(*======================================================================================================================================*)
(*fb_StringConvRB16F:	Zusammensetzen des Strings für 16Fach Bus Relaismodul		*)
(*
Date          	| Version    	| created under        	| Author          	| Remark *)
(*====================================================================================================================================================*)
(*08/05/2025   	| 1.00      		| TC3		  		| N.Kersting       | first release *)
(*====================================================================================================================================================*)
FUNCTION_BLOCK fb_StringConvRB16F
VAR_INPUT
	I_bReset			:BOOL;							(* Reset Befehl auslösen *)
	I_bRedLEDOn			:BOOL;							(* Schaltet nur die Rote Modul LED ein*)
	I_bRedLEDOff		:BOOL;							(* Schaltet nur die Rote Modul LED aus*)
	I_diID				:DINT;							(* Device ID *)
	I_bOut    	 		:ARRAY[1..16] OF BOOL;     	  	(* gewünschter Relais zustand (TRUE = An %)*)
	
	I_iSection			:INT :=1;							(* Paarweise Schalten 1= 1&2 2= 3&4 usw. *)
	
	I_sStartZeichen		:BYTE := 16#FD;					(* Startzeichen Präfix *)
	I_sEndZeichen		:BYTE := 16#FE;					(* Endzeichen Suffix *)
END_VAR
VAR_OUTPUT
	Q_sConvString		:STRING(255);
END_VAR
VAR
	iStartOut			:INT := 1;
	iStartInstIDExt		:INT :=65;
	
END_VAR

IF NOT I_bReset
THEN
	IF I_bRedLEDOn
	THEN
		(* Rote Modul LED Ein*)
		iStartInstIDExt := 210;
		
		Q_sConvString:=	CONCAT(F_ToCHR(I_sStartZeichen),DINT_TO_STRING(I_diID));
		Q_sConvString:=	CONCAT(Q_sConvString,'.OUT.');
		Q_sConvString:=	CONCAT(Q_sConvString,INT_TO_STRING(iStartInstIDExt));
		Q_sConvString:=	CONCAT(Q_sConvString,'.ON');
		Q_sConvString:=	CONCAT(Q_sConvString,F_ToCHR(I_sEndZeichen));
	ELSIF
		I_bRedLEDOff
	THEN
		(* Rote Modul LED Aus*)
		iStartInstIDExt := 210;
		
		Q_sConvString:=	CONCAT(F_ToCHR(I_sStartZeichen),DINT_TO_STRING(I_diID));
		Q_sConvString:=	CONCAT(Q_sConvString,'.OUT.');
		Q_sConvString:=	CONCAT(Q_sConvString,INT_TO_STRING(iStartInstIDExt));
		Q_sConvString:=	CONCAT(Q_sConvString,'.OFF');
		Q_sConvString:=	CONCAT(Q_sConvString,F_ToCHR(I_sEndZeichen));
	ELSE
		CASE I_iSection OF
			
		0:	Q_sConvString:='';
		
		1:	(* 1 & 2 Schalten *)
			iStartInstIDExt := 17;
			iStartOut :=	1;
			
			Q_sConvString:=	CONCAT(F_ToCHR(I_sStartZeichen),DINT_TO_STRING(I_diID));
			Q_sConvString:=	CONCAT(Q_sConvString,'.OUT.');
			Q_sConvString:=	CONCAT(Q_sConvString,INT_TO_STRING(iStartInstIDExt));
			IF I_bOut[iStartOut]
			THEN
				Q_sConvString:=	CONCAT(Q_sConvString,'.ON');
			ELSE
				Q_sConvString:=	CONCAT(Q_sConvString,'.OFF');
			END_IF
			Q_sConvString:=	CONCAT(Q_sConvString,F_ToCHR(I_sEndZeichen));
			
			(* ##2 ##*)
			iStartInstIDExt := iStartInstIDExt +1;
			iStartOut:= iStartOut+1;
			
			Q_sConvString:=	CONCAT(Q_sConvString,F_ToCHR(I_sStartZeichen));
			Q_sConvString:=	CONCAT(Q_sConvString,DINT_TO_STRING(I_diID));
			Q_sConvString:=	CONCAT(Q_sConvString,'.OUT.');
			Q_sConvString:=	CONCAT(Q_sConvString,INT_TO_STRING(iStartInstIDExt));
			IF I_bOut[iStartOut]
			THEN
				Q_sConvString:=	CONCAT(Q_sConvString,'.ON');
			ELSE
				Q_sConvString:=	CONCAT(Q_sConvString,'.OFF');
			END_IF
			Q_sConvString:=	CONCAT(Q_sConvString,F_ToCHR(I_sEndZeichen));
		
			(* ##3 ##*)
			iStartInstIDExt := iStartInstIDExt +1;
			iStartOut:= iStartOut+1;
			
			Q_sConvString:=	CONCAT(Q_sConvString,F_ToCHR(I_sStartZeichen));
			Q_sConvString:=	CONCAT(Q_sConvString,DINT_TO_STRING(I_diID));
			Q_sConvString:=	CONCAT(Q_sConvString,'.OUT.');
			Q_sConvString:=	CONCAT(Q_sConvString,INT_TO_STRING(iStartInstIDExt));
			IF I_bOut[iStartOut]
			THEN
				Q_sConvString:=	CONCAT(Q_sConvString,'.ON');
			ELSE
				Q_sConvString:=	CONCAT(Q_sConvString,'.OFF');
			END_IF
			Q_sConvString:=	CONCAT(Q_sConvString,F_ToCHR(I_sEndZeichen));
			
			(* ##4 ##*)
			iStartInstIDExt := iStartInstIDExt +1;
			iStartOut:= iStartOut+1;
			
			Q_sConvString:=	CONCAT(Q_sConvString,F_ToCHR(I_sStartZeichen));
			Q_sConvString:=	CONCAT(Q_sConvString,DINT_TO_STRING(I_diID));
			Q_sConvString:=	CONCAT(Q_sConvString,'.OUT.');
			Q_sConvString:=	CONCAT(Q_sConvString,INT_TO_STRING(iStartInstIDExt));
			IF I_bOut[iStartOut]
			THEN
				Q_sConvString:=	CONCAT(Q_sConvString,'.ON');
			ELSE
				Q_sConvString:=	CONCAT(Q_sConvString,'.OFF');
			END_IF
			Q_sConvString:=	CONCAT(Q_sConvString,F_ToCHR(I_sEndZeichen));
		
			(* ##5 ##*)
			iStartInstIDExt := iStartInstIDExt +1;
			iStartOut:= iStartOut+1;
			
			Q_sConvString:=	CONCAT(Q_sConvString,F_ToCHR(I_sStartZeichen));
			Q_sConvString:=	CONCAT(Q_sConvString,DINT_TO_STRING(I_diID));
			Q_sConvString:=	CONCAT(Q_sConvString,'.OUT.');
			Q_sConvString:=	CONCAT(Q_sConvString,INT_TO_STRING(iStartInstIDExt));
			IF I_bOut[iStartOut]
			THEN
				Q_sConvString:=	CONCAT(Q_sConvString,'.ON');
			ELSE
				Q_sConvString:=	CONCAT(Q_sConvString,'.OFF');
			END_IF
			Q_sConvString:=	CONCAT(Q_sConvString,F_ToCHR(I_sEndZeichen));
			
			(* ##6 ##*)
			iStartInstIDExt := iStartInstIDExt +1;
			iStartOut:= iStartOut+1;
			
			Q_sConvString:=	CONCAT(Q_sConvString,F_ToCHR(I_sStartZeichen));
			Q_sConvString:=	CONCAT(Q_sConvString,DINT_TO_STRING(I_diID));
			Q_sConvString:=	CONCAT(Q_sConvString,'.OUT.');
			Q_sConvString:=	CONCAT(Q_sConvString,INT_TO_STRING(iStartInstIDExt));
			IF I_bOut[iStartOut]
			THEN
				Q_sConvString:=	CONCAT(Q_sConvString,'.ON');
			ELSE
				Q_sConvString:=	CONCAT(Q_sConvString,'.OFF');
			END_IF
			Q_sConvString:=	CONCAT(Q_sConvString,F_ToCHR(I_sEndZeichen));
		
			(* ##7 ##*)
			iStartInstIDExt := iStartInstIDExt +1;
			iStartOut:= iStartOut+1;
			
			Q_sConvString:=	CONCAT(Q_sConvString,F_ToCHR(I_sStartZeichen));
			Q_sConvString:=	CONCAT(Q_sConvString,DINT_TO_STRING(I_diID));
			Q_sConvString:=	CONCAT(Q_sConvString,'.OUT.');
			Q_sConvString:=	CONCAT(Q_sConvString,INT_TO_STRING(iStartInstIDExt));
			IF I_bOut[iStartOut]
			THEN
				Q_sConvString:=	CONCAT(Q_sConvString,'.ON');
			ELSE
				Q_sConvString:=	CONCAT(Q_sConvString,'.OFF');
			END_IF
			Q_sConvString:=	CONCAT(Q_sConvString,F_ToCHR(I_sEndZeichen));
			
			(* ##8 ##*)
			iStartInstIDExt := iStartInstIDExt +1;
			iStartOut:= iStartOut+1;
			
			Q_sConvString:=	CONCAT(Q_sConvString,F_ToCHR(I_sStartZeichen));
			Q_sConvString:=	CONCAT(Q_sConvString,DINT_TO_STRING(I_diID));
			Q_sConvString:=	CONCAT(Q_sConvString,'.OUT.');
			Q_sConvString:=	CONCAT(Q_sConvString,INT_TO_STRING(iStartInstIDExt));
			IF I_bOut[iStartOut]
			THEN
				Q_sConvString:=	CONCAT(Q_sConvString,'.ON');
			ELSE
				Q_sConvString:=	CONCAT(Q_sConvString,'.OFF');
			END_IF
			Q_sConvString:=	CONCAT(Q_sConvString,F_ToCHR(I_sEndZeichen));
		
		2:	(* 9 & 10 Schalten *)
			iStartInstIDExt := 33;
			iStartOut :=	9;
			
			Q_sConvString:=	CONCAT(F_ToCHR(I_sStartZeichen),DINT_TO_STRING(I_diID));
			Q_sConvString:=	CONCAT(Q_sConvString,'.OUT.');
			Q_sConvString:=	CONCAT(Q_sConvString,INT_TO_STRING(iStartInstIDExt));
			IF I_bOut[iStartOut]
			THEN
				Q_sConvString:=	CONCAT(Q_sConvString,'.ON');
			ELSE
				Q_sConvString:=	CONCAT(Q_sConvString,'.OFF');
			END_IF
			Q_sConvString:=	CONCAT(Q_sConvString,F_ToCHR(I_sEndZeichen));
			
			(* ##10 ##*)
			iStartInstIDExt := iStartInstIDExt +1;
			iStartOut:= iStartOut+1;
			
			Q_sConvString:=	CONCAT(Q_sConvString,F_ToCHR(I_sStartZeichen));
			Q_sConvString:=	CONCAT(Q_sConvString,DINT_TO_STRING(I_diID));
			Q_sConvString:=	CONCAT(Q_sConvString,'.OUT.');
			Q_sConvString:=	CONCAT(Q_sConvString,INT_TO_STRING(iStartInstIDExt));
			IF I_bOut[iStartOut]
			THEN
				Q_sConvString:=	CONCAT(Q_sConvString,'.ON');
			ELSE
				Q_sConvString:=	CONCAT(Q_sConvString,'.OFF');
			END_IF
			Q_sConvString:=	CONCAT(Q_sConvString,F_ToCHR(I_sEndZeichen));
		
			(* ##11 ##*)
			iStartInstIDExt := iStartInstIDExt +1;
			iStartOut:= iStartOut+1;
			
			Q_sConvString:=	CONCAT(Q_sConvString,F_ToCHR(I_sStartZeichen));
			Q_sConvString:=	CONCAT(Q_sConvString,DINT_TO_STRING(I_diID));
			Q_sConvString:=	CONCAT(Q_sConvString,'.OUT.');
			Q_sConvString:=	CONCAT(Q_sConvString,INT_TO_STRING(iStartInstIDExt));
			IF I_bOut[iStartOut]
			THEN
				Q_sConvString:=	CONCAT(Q_sConvString,'.ON');
			ELSE
				Q_sConvString:=	CONCAT(Q_sConvString,'.OFF');
			END_IF
			Q_sConvString:=	CONCAT(Q_sConvString,F_ToCHR(I_sEndZeichen));
			
			(* ##12 ##*)
			iStartInstIDExt := iStartInstIDExt +1;
			iStartOut:= iStartOut+1;
			
			Q_sConvString:=	CONCAT(Q_sConvString,F_ToCHR(I_sStartZeichen));
			Q_sConvString:=	CONCAT(Q_sConvString,DINT_TO_STRING(I_diID));
			Q_sConvString:=	CONCAT(Q_sConvString,'.OUT.');
			Q_sConvString:=	CONCAT(Q_sConvString,INT_TO_STRING(iStartInstIDExt));
			IF I_bOut[iStartOut]
			THEN
				Q_sConvString:=	CONCAT(Q_sConvString,'.ON');
			ELSE
				Q_sConvString:=	CONCAT(Q_sConvString,'.OFF');
			END_IF
			Q_sConvString:=	CONCAT(Q_sConvString,F_ToCHR(I_sEndZeichen));
		
			(* ##13 ##*)
			iStartInstIDExt := iStartInstIDExt +1;
			iStartOut:= iStartOut+1;
			
			Q_sConvString:=	CONCAT(Q_sConvString,F_ToCHR(I_sStartZeichen));
			Q_sConvString:=	CONCAT(Q_sConvString,DINT_TO_STRING(I_diID));
			Q_sConvString:=	CONCAT(Q_sConvString,'.OUT.');
			Q_sConvString:=	CONCAT(Q_sConvString,INT_TO_STRING(iStartInstIDExt));
			IF I_bOut[iStartOut]
			THEN
				Q_sConvString:=	CONCAT(Q_sConvString,'.ON');
			ELSE
				Q_sConvString:=	CONCAT(Q_sConvString,'.OFF');
			END_IF
			Q_sConvString:=	CONCAT(Q_sConvString,F_ToCHR(I_sEndZeichen));
			
			(* ##14 ##*)
			iStartInstIDExt := iStartInstIDExt +1;
			iStartOut:= iStartOut+1;
			
			Q_sConvString:=	CONCAT(Q_sConvString,F_ToCHR(I_sStartZeichen));
			Q_sConvString:=	CONCAT(Q_sConvString,DINT_TO_STRING(I_diID));
			Q_sConvString:=	CONCAT(Q_sConvString,'.OUT.');
			Q_sConvString:=	CONCAT(Q_sConvString,INT_TO_STRING(iStartInstIDExt));
			IF I_bOut[iStartOut]
			THEN
				Q_sConvString:=	CONCAT(Q_sConvString,'.ON');
			ELSE
				Q_sConvString:=	CONCAT(Q_sConvString,'.OFF');
			END_IF
			Q_sConvString:=	CONCAT(Q_sConvString,F_ToCHR(I_sEndZeichen));
		
			(* ##15 ##*)
			iStartInstIDExt := iStartInstIDExt +1;
			iStartOut:= iStartOut+1;
			
			Q_sConvString:=	CONCAT(Q_sConvString,F_ToCHR(I_sStartZeichen));
			Q_sConvString:=	CONCAT(Q_sConvString,DINT_TO_STRING(I_diID));
			Q_sConvString:=	CONCAT(Q_sConvString,'.OUT.');
			Q_sConvString:=	CONCAT(Q_sConvString,INT_TO_STRING(iStartInstIDExt));
			IF I_bOut[iStartOut]
			THEN
				Q_sConvString:=	CONCAT(Q_sConvString,'.ON');
			ELSE
				Q_sConvString:=	CONCAT(Q_sConvString,'.OFF');
			END_IF
			Q_sConvString:=	CONCAT(Q_sConvString,F_ToCHR(I_sEndZeichen));
			
			(* ##16 ##*)
			iStartInstIDExt := iStartInstIDExt +1;
			iStartOut:= iStartOut+1;
			
			Q_sConvString:=	CONCAT(Q_sConvString,F_ToCHR(I_sStartZeichen));
			Q_sConvString:=	CONCAT(Q_sConvString,DINT_TO_STRING(I_diID));
			Q_sConvString:=	CONCAT(Q_sConvString,'.OUT.');
			Q_sConvString:=	CONCAT(Q_sConvString,INT_TO_STRING(iStartInstIDExt));
			IF I_bOut[iStartOut]
			THEN
				Q_sConvString:=	CONCAT(Q_sConvString,'.ON');
			ELSE
				Q_sConvString:=	CONCAT(Q_sConvString,'.OFF');
			END_IF
			Q_sConvString:=	CONCAT(Q_sConvString,F_ToCHR(I_sEndZeichen));
		END_CASE
	END_IF
	
ELSE
	(* Reset *)
	Q_sConvString:=	CONCAT(F_ToCHR(I_sStartZeichen),DINT_TO_STRING(I_diID));
	Q_sConvString:=	CONCAT(Q_sConvString,'.SYS.');
	Q_sConvString:=	CONCAT(Q_sConvString,INT_TO_STRING(1));
	Q_sConvString:=	CONCAT(Q_sConvString,'.RESET');
	Q_sConvString:=	CONCAT(Q_sConvString,F_ToCHR(I_sEndZeichen));
END_IF

END_FUNCTION_BLOCK

(* stored: Version 1.1.0.1, ProductVersion 3.1.4024.12
   POU fb_StringConvRB16F: Id {e8a09989-e90a-48c9-b77f-5f391bcac87a}, SpecialFunc None *)
